// SIMATIC S7-200 SMART project (STEP 7-Micro/WIN SMART), CPU ST40

SYMBOL_TABLE Table 1
Start_SW         I0.3
Stop_SW          I0.4
Memory           M0.0
Level_1          I0.0
Level_2          I0.1
Level_3          I0.2
Liquid_1_Inlet   Q0.0
Liquid_2_Inlet   Q0.1
Mixer_Motor      Q0.3
Mixing_Timer     T101
Outlet_Valve     Q0.2
END_SYMBOL_TABLE

ORGANIZATION_BLOCK MAIN:OB1
TITLE=Program Comments
BEGIN
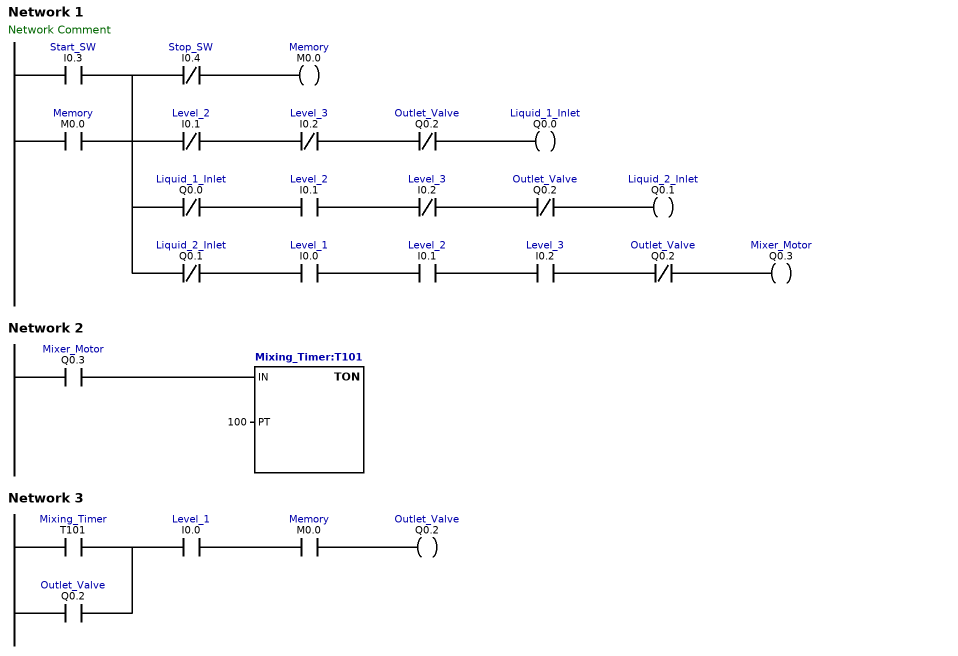
Network 1
// Network Comment
LD     Start_SW:I0.3
O      Memory:M0.0
LPS
AN     Stop_SW:I0.4
=      Memory:M0.0
LRD
AN     Level_2:I0.1
AN     Level_3:I0.2
AN     Outlet_Valve:Q0.2
=      Liquid_1_Inlet:Q0.0
LRD
AN     Liquid_1_Inlet:Q0.0
A      Level_2:I0.1
AN     Level_3:I0.2
AN     Outlet_Valve:Q0.2
=      Liquid_2_Inlet:Q0.1
LPP
AN     Liquid_2_Inlet:Q0.1
A      Level_1:I0.0
A      Level_2:I0.1
A      Level_3:I0.2
AN     Outlet_Valve:Q0.2
=      Mixer_Motor:Q0.3
Network 2
LD     Mixer_Motor:Q0.3
TON    Mixing_Timer:T101, 100
Network 3
LD     Mixing_Timer:T101
O      Outlet_Valve:Q0.2
A      Level_1:I0.0
A      Memory:M0.0
=      Outlet_Valve:Q0.2
END_ORGANIZATION_BLOCK
